FUNCTION Concat3 : T_MaxString
VAR_INPUT
	sExpression1: T_maxString;
	sExpression2: T_maxString;
	sExpression3: T_maxString;
END_VAR

Concat3 := CONCAT(sExpression1, sExpression2);
Concat3 := CONCAT(Concat3, sExpression3);

END_FUNCTION

(* stored: Version 1.1.0.1
   POU Concat3: Id {d708717a-7d4b-4e71-9714-b0ef0230c552}, SpecialFunc None *)
